// TIA Portal V17 export
// export: Created 2024-09-02T12:50:19.4817416Z, ExportSetting WithDefaults, DisplayName Totally Integrated Automation Portal, DisplayVersion V17, DisplayName TIA Portal Openness, DisplayVersion V17, DisplayName TIA Portal Version Control Interface, DisplayVersion V17, DisplayName STEP 7 Professional, DisplayVersion V17, DisplayName STEP 7 Safety, DisplayVersion V17, DisplayName WinCC Professional, DisplayVersion V17
FUNCTION "AnwFC_Omron_OP70_2" : Void   // FC190, LAD
{ S7_Optimized_Access := 'TRUE' }
VERSION : 0.1
// stored: AutoNumber false, IsIECCheckEnabled false, SetENOAutomatically false, UDAEnableTagReadback false
   VAR_TEMP
      tVKE0 : Bool;
      tVKE1 : Bool;
      tAuto : Bool;
      tHand : Bool;
      Motion_Release : Bool;
      t_dummy : Bool;
      tHmiBld : Bool;
      tHmiEnbl : Bool;
      tCnt : Int;
      tBAmode : Int;
      tHmiScreen : Bool;
      tHmiRelease : Bool;
      i : Int;
   END_VAR
   VAR_TEMP   // added for the SCL form of the ladder/FBD networks
      _w1 : Bool;
   END_VAR
BEGIN

REGION Network 1: ############# Moving Data To DB ###############
END_REGION

REGION Network 2: Copy Output
END_REGION

REGION Network 3: Copy Input
END_REGION

REGION Network 4: ############# Start Up Conditions ###############
END_REGION

REGION Network 5: VKE0/1
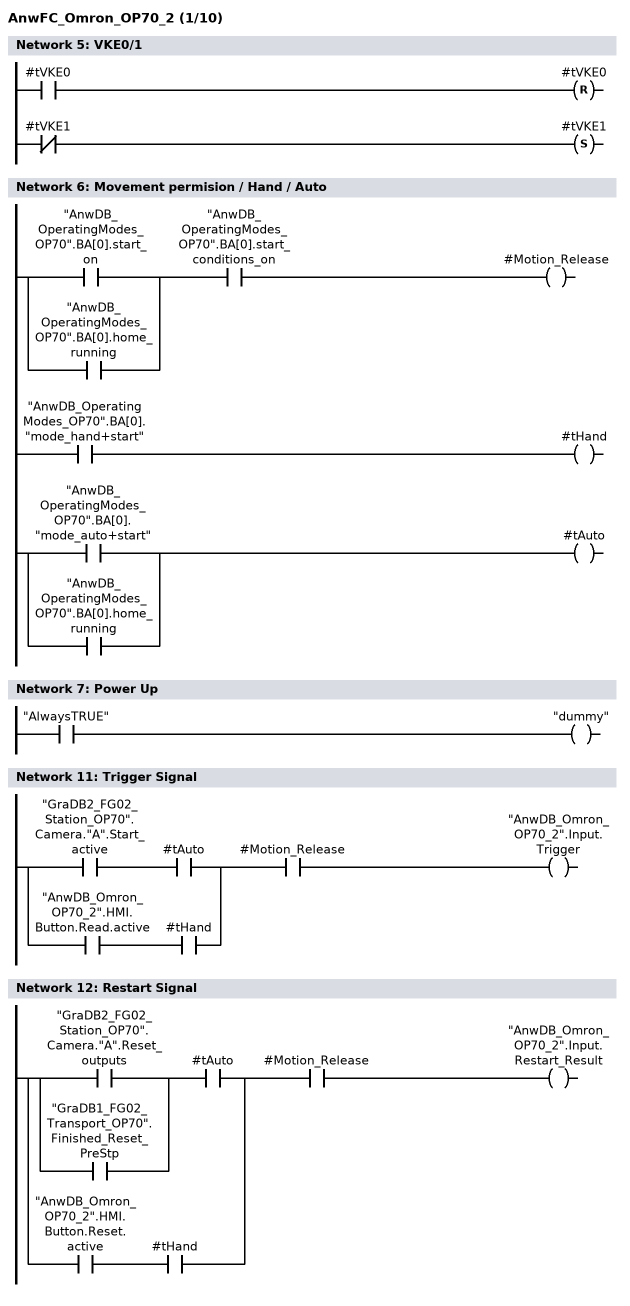
   RUNG wire#powerrail
      Contact( #tVKE0 )
      R_Coil( #tVKE0 )
   END_RUNG
   RUNG wire#powerrail
      I_Contact( #tVKE1 )
      S_Coil( #tVKE1 )
   END_RUNG
   // the same network as SCL:
   IF #tVKE0 THEN #tVKE0 := FALSE; END_IF;
   IF NOT #tVKE1 THEN #tVKE1 := TRUE; END_IF;
END_REGION

REGION Network 6: Movement permision / Hand / Auto
   RUNG wire#powerrail
      Contact( "AnwDB_OperatingModes_OP70".BA[0].start_on )
      wire#w1
      Contact( "AnwDB_OperatingModes_OP70".BA[0].start_conditions_on )
      Coil( #Motion_Release )
   END_RUNG
   RUNG wire#powerrail
      Contact( "AnwDB_OperatingModes_OP70".BA[0].home_running )
   END_RUNG wire#w1
   RUNG wire#powerrail
      Contact( "AnwDB_OperatingModes_OP70".BA[0]."mode_hand+start" )
      Coil( #tHand )
   END_RUNG
   RUNG wire#powerrail
      Contact( "AnwDB_OperatingModes_OP70".BA[0]."mode_auto+start" )
      wire#w2
      Coil( #tAuto )
   END_RUNG
   RUNG wire#powerrail
      Contact( "AnwDB_OperatingModes_OP70".BA[0].home_running )
   END_RUNG wire#w2
   // the same network as SCL:
   #Motion_Release := ("AnwDB_OperatingModes_OP70".BA[0].start_on OR "AnwDB_OperatingModes_OP70".BA[0].home_running) AND "AnwDB_OperatingModes_OP70".BA[0].start_conditions_on;
   #tHand := "AnwDB_OperatingModes_OP70".BA[0]."mode_hand+start";
   #tAuto := "AnwDB_OperatingModes_OP70".BA[0]."mode_auto+start" OR "AnwDB_OperatingModes_OP70".BA[0].home_running;
END_REGION

REGION Network 7: Power Up
   RUNG wire#powerrail
      Contact( "AlwaysTRUE" )
      Coil( "dummy" )
   END_RUNG
   // the same network as SCL:
   "dummy" := "AlwaysTRUE";
END_REGION

REGION Network 8: ############# Data Operation ###############
END_REGION

REGION Network 9: Copy ID number
END_REGION

REGION Network 10: ############# Program Selection And Start ###############
END_REGION

REGION Network 11: Trigger Signal
   RUNG wire#powerrail
      Contact( "GraDB2_FG02_Station_OP70".Camera."A".Start_active )
      Contact( #tAuto )
      wire#w1
      Contact( #Motion_Release )
      Coil( "AnwDB_Omron_OP70_2".Input.Trigger )
   END_RUNG
   RUNG wire#powerrail
      Contact( "AnwDB_Omron_OP70_2".HMI.Button.Read.active )
      Contact( #tHand )
   END_RUNG wire#w1
   // the same network as SCL:
   "AnwDB_Omron_OP70_2".Input.Trigger := (("GraDB2_FG02_Station_OP70".Camera."A".Start_active AND #tAuto) OR ("AnwDB_Omron_OP70_2".HMI.Button.Read.active AND #tHand)) AND #Motion_Release;
END_REGION

REGION Network 12: Restart Signal
   RUNG wire#powerrail
      Contact( "GraDB2_FG02_Station_OP70".Camera."A".Reset_outputs )
      wire#w1
      Contact( #tAuto )
      wire#w2
      Contact( #Motion_Release )
      Coil( "AnwDB_Omron_OP70_2".Input.Restart_Result )
   END_RUNG
   RUNG wire#powerrail
      Contact( "GraDB1_FG02_Transport_OP70".Finished_Reset_PreStp )
   END_RUNG wire#w1
   RUNG wire#powerrail
      Contact( "AnwDB_Omron_OP70_2".HMI.Button.Reset.active )
      Contact( #tHand )
   END_RUNG wire#w2
   // the same network as SCL:
   "AnwDB_Omron_OP70_2".Input.Restart_Result := ((("GraDB2_FG02_Station_OP70".Camera."A".Reset_outputs OR "GraDB1_FG02_Transport_OP70".Finished_Reset_PreStp) AND #tAuto) OR ("AnwDB_Omron_OP70_2".HMI.Button.Reset.active AND #tHand)) AND #Motion_Release;
END_REGION

REGION Network 13: Ack Signal
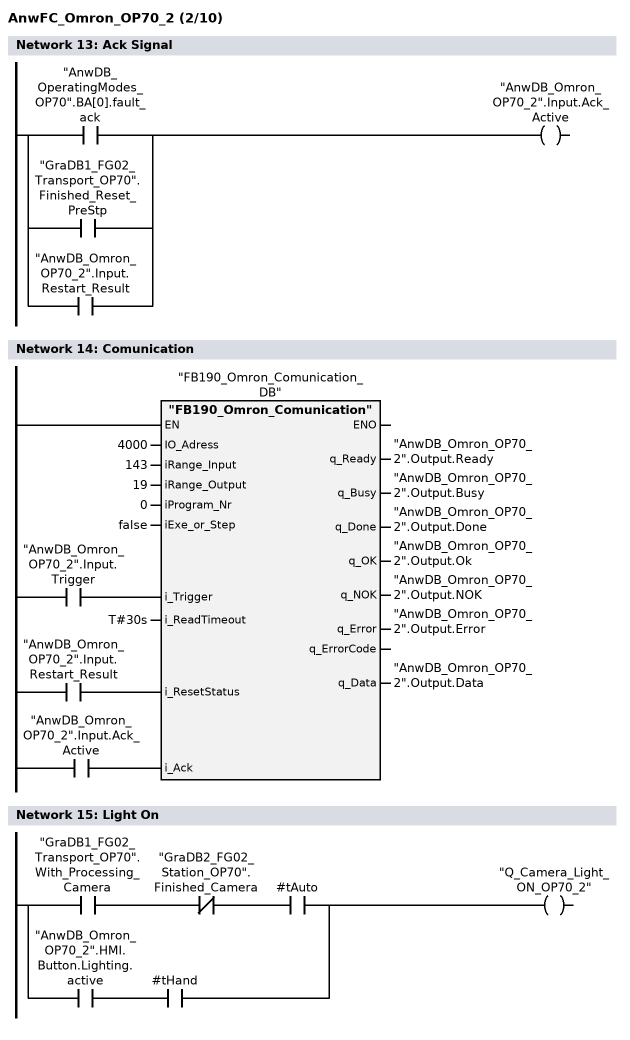
   RUNG wire#powerrail
      Contact( "AnwDB_OperatingModes_OP70".BA[0].fault_ack )
      wire#w1
      Coil( "AnwDB_Omron_OP70_2".Input.Ack_Active )
   END_RUNG
   RUNG wire#powerrail
      Contact( "GraDB1_FG02_Transport_OP70".Finished_Reset_PreStp )
   END_RUNG wire#w1
   RUNG wire#powerrail
      Contact( "AnwDB_Omron_OP70_2".Input.Restart_Result )
   END_RUNG wire#w1
   // the same network as SCL:
   "AnwDB_Omron_OP70_2".Input.Ack_Active := "AnwDB_OperatingModes_OP70".BA[0].fault_ack OR "GraDB1_FG02_Transport_OP70".Finished_Reset_PreStp OR "AnwDB_Omron_OP70_2".Input.Restart_Result;
END_REGION

REGION Network 14: Comunication
   RUNG wire#powerrail
      "FB190_Omron_Comunication_DB"(i_Trigger := wire#w1, i_ResetStatus := wire#w2, i_Ack := wire#w3, IO_Adress := 4000, iRange_Input := 143, iRange_Output := 19, iProgram_Nr := 0, iExe_or_Step := false, i_ReadTimeout := T#30s, q_Ready => "AnwDB_Omron_OP70_2".Output.Ready, q_Busy => "AnwDB_Omron_OP70_2".Output.Busy, q_Done => "AnwDB_Omron_OP70_2".Output.Done, q_OK => "AnwDB_Omron_OP70_2".Output.Ok, q_NOK => "AnwDB_Omron_OP70_2".Output.NOK, q_Error => "AnwDB_Omron_OP70_2".Output.Error, q_ErrorCode =>, q_Data => "AnwDB_Omron_OP70_2".Output.Data)
   END_RUNG
   RUNG wire#powerrail
      Contact( "AnwDB_Omron_OP70_2".Input.Trigger )
   END_RUNG wire#w1
   RUNG wire#powerrail
      Contact( "AnwDB_Omron_OP70_2".Input.Restart_Result )
   END_RUNG wire#w2
   RUNG wire#powerrail
      Contact( "AnwDB_Omron_OP70_2".Input.Ack_Active )
   END_RUNG wire#w3
   // the same network as SCL:
   "FB190_Omron_Comunication_DB"(IO_Adress := 4000,   // "FB190_Omron_Comunication"
                           iRange_Input := 143,
                           iRange_Output := 19,
                           iProgram_Nr := 0,
                           iExe_or_Step := false,
                           i_Trigger := "AnwDB_Omron_OP70_2".Input.Trigger,
                           i_ReadTimeout := T#30s,
                           i_ResetStatus := "AnwDB_Omron_OP70_2".Input.Restart_Result,
                           i_Ack := "AnwDB_Omron_OP70_2".Input.Ack_Active,
                           q_Ready => "AnwDB_Omron_OP70_2".Output.Ready,
                           q_Busy => "AnwDB_Omron_OP70_2".Output.Busy,
                           q_Done => "AnwDB_Omron_OP70_2".Output.Done,
                           q_OK => "AnwDB_Omron_OP70_2".Output.Ok,
                           q_NOK => "AnwDB_Omron_OP70_2".Output.NOK,
                           q_Error => "AnwDB_Omron_OP70_2".Output.Error,
                           q_Data => "AnwDB_Omron_OP70_2".Output.Data);
END_REGION

REGION Network 15: Light On
   RUNG wire#powerrail
      Contact( "GraDB1_FG02_Transport_OP70".With_Processing_Camera )
      I_Contact( "GraDB2_FG02_Station_OP70".Finished_Camera )
      Contact( #tAuto )
      wire#w1
      Coil( "Q_Camera_Light_ON_OP70_2" )
   END_RUNG
   RUNG wire#powerrail
      Contact( "AnwDB_Omron_OP70_2".HMI.Button.Lighting.active )
      Contact( #tHand )
   END_RUNG wire#w1
   // the same network as SCL:
   "Q_Camera_Light_ON_OP70_2" := ("GraDB1_FG02_Transport_OP70".With_Processing_Camera AND NOT "GraDB2_FG02_Station_OP70".Finished_Camera AND #tAuto) OR ("AnwDB_Omron_OP70_2".HMI.Button.Lighting.active AND #tHand);
END_REGION

REGION Network 16: ############# Program Status ###############
END_REGION

REGION Network 17: BEA[1].Ebit[1] - Damper 1 OP 50
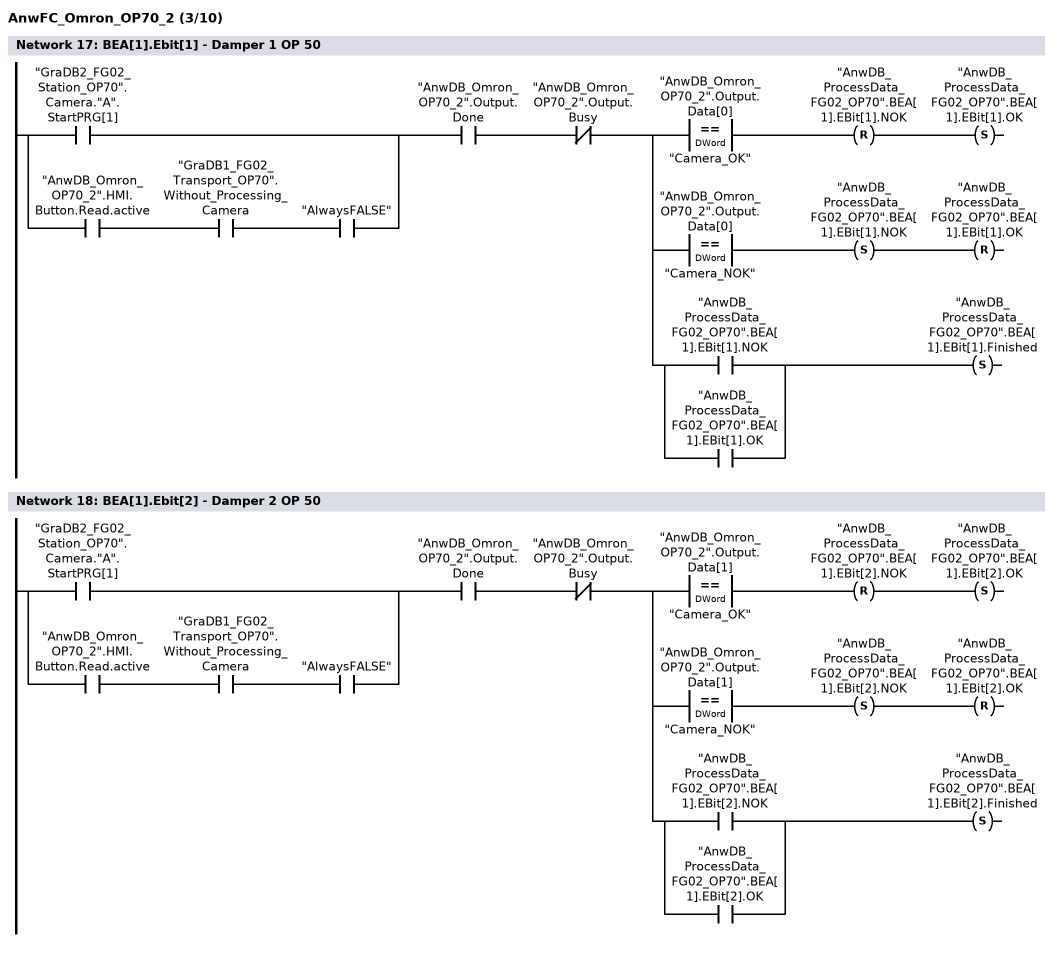
   RUNG wire#powerrail
      Contact( "GraDB2_FG02_Station_OP70".Camera."A".StartPRG[1] )
      wire#w1
      Contact( "AnwDB_Omron_OP70_2".Output.Done )
      I_Contact( "AnwDB_Omron_OP70_2".Output.Busy )
      wire#w2
      { S7_Templates := "SrcType := DWord" } EQ_Contact(in1 := "AnwDB_Omron_OP70_2".Output.Data[0], in2 := "Camera_OK")
      R_Coil( "AnwDB_ProcessData_FG02_OP70".BEA[1].EBit[1].NOK )
      S_Coil( "AnwDB_ProcessData_FG02_OP70".BEA[1].EBit[1].OK )
   END_RUNG
   RUNG wire#powerrail
      Contact( "AnwDB_Omron_OP70_2".HMI.Button.Read.active )
      Contact( "GraDB1_FG02_Transport_OP70".Without_Processing_Camera )
      Contact( "AlwaysFALSE" )
   END_RUNG wire#w1
   RUNG wire#w2
      { S7_Templates := "SrcType := DWord" } EQ_Contact(in1 := "AnwDB_Omron_OP70_2".Output.Data[0], in2 := "Camera_NOK")
      S_Coil( "AnwDB_ProcessData_FG02_OP70".BEA[1].EBit[1].NOK )
      R_Coil( "AnwDB_ProcessData_FG02_OP70".BEA[1].EBit[1].OK )
   END_RUNG
   RUNG wire#w2
      Contact( "AnwDB_ProcessData_FG02_OP70".BEA[1].EBit[1].NOK )
      wire#w3
      S_Coil( "AnwDB_ProcessData_FG02_OP70".BEA[1].EBit[1].Finished )
   END_RUNG
   RUNG wire#w2
      Contact( "AnwDB_ProcessData_FG02_OP70".BEA[1].EBit[1].OK )
   END_RUNG wire#w3
   // the same network as SCL:
   #_w1 := ("GraDB2_FG02_Station_OP70".Camera."A".StartPRG[1] OR ("AnwDB_Omron_OP70_2".HMI.Button.Read.active AND "GraDB1_FG02_Transport_OP70".Without_Processing_Camera AND "AlwaysFALSE")) AND "AnwDB_Omron_OP70_2".Output.Done AND NOT "AnwDB_Omron_OP70_2".Output.Busy;
   IF #_w1 AND ("AnwDB_Omron_OP70_2".Output.Data[0] = "Camera_OK") THEN
       "AnwDB_ProcessData_FG02_OP70".BEA[1].EBit[1].NOK := FALSE;
       "AnwDB_ProcessData_FG02_OP70".BEA[1].EBit[1].OK := TRUE;
   END_IF;
   IF #_w1 AND ("AnwDB_Omron_OP70_2".Output.Data[0] = "Camera_NOK") THEN
       "AnwDB_ProcessData_FG02_OP70".BEA[1].EBit[1].NOK := TRUE;
       "AnwDB_ProcessData_FG02_OP70".BEA[1].EBit[1].OK := FALSE;
   END_IF;
   IF #_w1 AND ("AnwDB_ProcessData_FG02_OP70".BEA[1].EBit[1].NOK OR "AnwDB_ProcessData_FG02_OP70".BEA[1].EBit[1].OK) THEN
       "AnwDB_ProcessData_FG02_OP70".BEA[1].EBit[1].Finished := TRUE;
   END_IF;
END_REGION

REGION Network 18: BEA[1].Ebit[2] - Damper 2 OP 50
   RUNG wire#powerrail
      Contact( "GraDB2_FG02_Station_OP70".Camera."A".StartPRG[1] )
      wire#w1
      Contact( "AnwDB_Omron_OP70_2".Output.Done )
      I_Contact( "AnwDB_Omron_OP70_2".Output.Busy )
      wire#w2
      { S7_Templates := "SrcType := DWord" } EQ_Contact(in1 := "AnwDB_Omron_OP70_2".Output.Data[1], in2 := "Camera_OK")
      R_Coil( "AnwDB_ProcessData_FG02_OP70".BEA[1].EBit[2].NOK )
      S_Coil( "AnwDB_ProcessData_FG02_OP70".BEA[1].EBit[2].OK )
   END_RUNG
   RUNG wire#powerrail
      Contact( "AnwDB_Omron_OP70_2".HMI.Button.Read.active )
      Contact( "GraDB1_FG02_Transport_OP70".Without_Processing_Camera )
      Contact( "AlwaysFALSE" )
   END_RUNG wire#w1
   RUNG wire#w2
      { S7_Templates := "SrcType := DWord" } EQ_Contact(in1 := "AnwDB_Omron_OP70_2".Output.Data[1], in2 := "Camera_NOK")
      S_Coil( "AnwDB_ProcessData_FG02_OP70".BEA[1].EBit[2].NOK )
      R_Coil( "AnwDB_ProcessData_FG02_OP70".BEA[1].EBit[2].OK )
   END_RUNG
   RUNG wire#w2
      Contact( "AnwDB_ProcessData_FG02_OP70".BEA[1].EBit[2].NOK )
      wire#w3
      S_Coil( "AnwDB_ProcessData_FG02_OP70".BEA[1].EBit[2].Finished )
   END_RUNG
   RUNG wire#w2
      Contact( "AnwDB_ProcessData_FG02_OP70".BEA[1].EBit[2].OK )
   END_RUNG wire#w3
   // the same network as SCL:
   #_w1 := ("GraDB2_FG02_Station_OP70".Camera."A".StartPRG[1] OR ("AnwDB_Omron_OP70_2".HMI.Button.Read.active AND "GraDB1_FG02_Transport_OP70".Without_Processing_Camera AND "AlwaysFALSE")) AND "AnwDB_Omron_OP70_2".Output.Done AND NOT "AnwDB_Omron_OP70_2".Output.Busy;
   IF #_w1 AND ("AnwDB_Omron_OP70_2".Output.Data[1] = "Camera_OK") THEN
       "AnwDB_ProcessData_FG02_OP70".BEA[1].EBit[2].NOK := FALSE;
       "AnwDB_ProcessData_FG02_OP70".BEA[1].EBit[2].OK := TRUE;
   END_IF;
   IF #_w1 AND ("AnwDB_Omron_OP70_2".Output.Data[1] = "Camera_NOK") THEN
       "AnwDB_ProcessData_FG02_OP70".BEA[1].EBit[2].NOK := TRUE;
       "AnwDB_ProcessData_FG02_OP70".BEA[1].EBit[2].OK := FALSE;
   END_IF;
   IF #_w1 AND ("AnwDB_ProcessData_FG02_OP70".BEA[1].EBit[2].NOK OR "AnwDB_ProcessData_FG02_OP70".BEA[1].EBit[2].OK) THEN
       "AnwDB_ProcessData_FG02_OP70".BEA[1].EBit[2].Finished := TRUE;
   END_IF;
END_REGION

REGION Network 19: BEA[1].Ebit[3] - Damper 3 OP 50
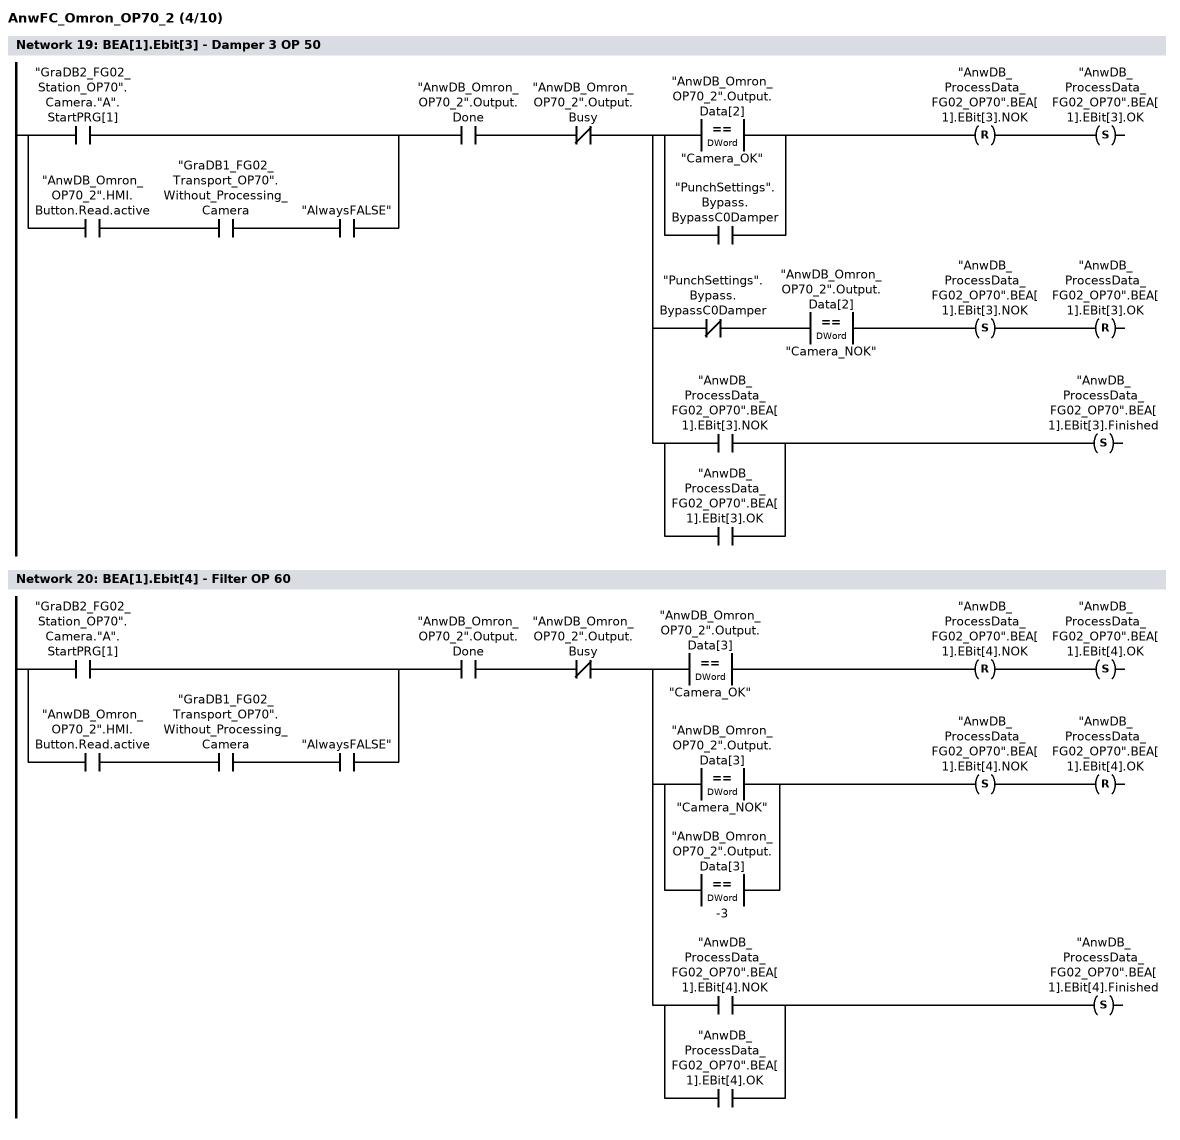
   RUNG wire#powerrail
      Contact( "GraDB2_FG02_Station_OP70".Camera."A".StartPRG[1] )
      wire#w1
      Contact( "AnwDB_Omron_OP70_2".Output.Done )
      I_Contact( "AnwDB_Omron_OP70_2".Output.Busy )
      wire#w2
      { S7_Templates := "SrcType := DWord" } EQ_Contact(in1 := "AnwDB_Omron_OP70_2".Output.Data[2], in2 := "Camera_OK")
      wire#w3
      R_Coil( "AnwDB_ProcessData_FG02_OP70".BEA[1].EBit[3].NOK )
      S_Coil( "AnwDB_ProcessData_FG02_OP70".BEA[1].EBit[3].OK )
   END_RUNG
   RUNG wire#powerrail
      Contact( "AnwDB_Omron_OP70_2".HMI.Button.Read.active )
      Contact( "GraDB1_FG02_Transport_OP70".Without_Processing_Camera )
      Contact( "AlwaysFALSE" )
   END_RUNG wire#w1
   RUNG wire#w2
      Contact( "PunchSettings".Bypass.BypassC0Damper )
   END_RUNG wire#w3
   RUNG wire#w2
      I_Contact( "PunchSettings".Bypass.BypassC0Damper )
      { S7_Templates := "SrcType := DWord" } EQ_Contact(in1 := "AnwDB_Omron_OP70_2".Output.Data[2], in2 := "Camera_NOK")
      S_Coil( "AnwDB_ProcessData_FG02_OP70".BEA[1].EBit[3].NOK )
      R_Coil( "AnwDB_ProcessData_FG02_OP70".BEA[1].EBit[3].OK )
   END_RUNG
   RUNG wire#w2
      Contact( "AnwDB_ProcessData_FG02_OP70".BEA[1].EBit[3].NOK )
      wire#w4
      S_Coil( "AnwDB_ProcessData_FG02_OP70".BEA[1].EBit[3].Finished )
   END_RUNG
   RUNG wire#w2
      Contact( "AnwDB_ProcessData_FG02_OP70".BEA[1].EBit[3].OK )
   END_RUNG wire#w4
   // the same network as SCL:
   #_w1 := ("GraDB2_FG02_Station_OP70".Camera."A".StartPRG[1] OR ("AnwDB_Omron_OP70_2".HMI.Button.Read.active AND "GraDB1_FG02_Transport_OP70".Without_Processing_Camera AND "AlwaysFALSE")) AND "AnwDB_Omron_OP70_2".Output.Done AND NOT "AnwDB_Omron_OP70_2".Output.Busy;
   IF #_w1 AND (("AnwDB_Omron_OP70_2".Output.Data[2] = "Camera_OK") OR "PunchSettings".Bypass.BypassC0Damper) THEN
       "AnwDB_ProcessData_FG02_OP70".BEA[1].EBit[3].NOK := FALSE;
       "AnwDB_ProcessData_FG02_OP70".BEA[1].EBit[3].OK := TRUE;
   END_IF;
   IF #_w1 AND NOT "PunchSettings".Bypass.BypassC0Damper AND ("AnwDB_Omron_OP70_2".Output.Data[2] = "Camera_NOK") THEN
       "AnwDB_ProcessData_FG02_OP70".BEA[1].EBit[3].NOK := TRUE;
       "AnwDB_ProcessData_FG02_OP70".BEA[1].EBit[3].OK := FALSE;
   END_IF;
   IF #_w1 AND ("AnwDB_ProcessData_FG02_OP70".BEA[1].EBit[3].NOK OR "AnwDB_ProcessData_FG02_OP70".BEA[1].EBit[3].OK) THEN
       "AnwDB_ProcessData_FG02_OP70".BEA[1].EBit[3].Finished := TRUE;
   END_IF;
END_REGION

REGION Network 20: BEA[1].Ebit[4] - Filter OP 60
   RUNG wire#powerrail
      Contact( "GraDB2_FG02_Station_OP70".Camera."A".StartPRG[1] )
      wire#w1
      Contact( "AnwDB_Omron_OP70_2".Output.Done )
      I_Contact( "AnwDB_Omron_OP70_2".Output.Busy )
      wire#w2
      { S7_Templates := "SrcType := DWord" } EQ_Contact(in1 := "AnwDB_Omron_OP70_2".Output.Data[3], in2 := "Camera_OK")
      R_Coil( "AnwDB_ProcessData_FG02_OP70".BEA[1].EBit[4].NOK )
      S_Coil( "AnwDB_ProcessData_FG02_OP70".BEA[1].EBit[4].OK )
   END_RUNG
   RUNG wire#powerrail
      Contact( "AnwDB_Omron_OP70_2".HMI.Button.Read.active )
      Contact( "GraDB1_FG02_Transport_OP70".Without_Processing_Camera )
      Contact( "AlwaysFALSE" )
   END_RUNG wire#w1
   RUNG wire#w2
      { S7_Templates := "SrcType := DWord" } EQ_Contact(in1 := "AnwDB_Omron_OP70_2".Output.Data[3], in2 := "Camera_NOK")
      wire#w3
      S_Coil( "AnwDB_ProcessData_FG02_OP70".BEA[1].EBit[4].NOK )
      R_Coil( "AnwDB_ProcessData_FG02_OP70".BEA[1].EBit[4].OK )
   END_RUNG
   RUNG wire#w2
      { S7_Templates := "SrcType := DWord" } EQ_Contact(in1 := "AnwDB_Omron_OP70_2".Output.Data[3], in2 := -3)
   END_RUNG wire#w3
   RUNG wire#w2
      Contact( "AnwDB_ProcessData_FG02_OP70".BEA[1].EBit[4].NOK )
      wire#w4
      S_Coil( "AnwDB_ProcessData_FG02_OP70".BEA[1].EBit[4].Finished )
   END_RUNG
   RUNG wire#w2
      Contact( "AnwDB_ProcessData_FG02_OP70".BEA[1].EBit[4].OK )
   END_RUNG wire#w4
   // the same network as SCL:
   #_w1 := ("GraDB2_FG02_Station_OP70".Camera."A".StartPRG[1] OR ("AnwDB_Omron_OP70_2".HMI.Button.Read.active AND "GraDB1_FG02_Transport_OP70".Without_Processing_Camera AND "AlwaysFALSE")) AND "AnwDB_Omron_OP70_2".Output.Done AND NOT "AnwDB_Omron_OP70_2".Output.Busy;
   IF #_w1 AND ("AnwDB_Omron_OP70_2".Output.Data[3] = "Camera_OK") THEN
       "AnwDB_ProcessData_FG02_OP70".BEA[1].EBit[4].NOK := FALSE;
       "AnwDB_ProcessData_FG02_OP70".BEA[1].EBit[4].OK := TRUE;
   END_IF;
   IF #_w1 AND (("AnwDB_Omron_OP70_2".Output.Data[3] = "Camera_NOK") OR ("AnwDB_Omron_OP70_2".Output.Data[3] = (-3))) THEN
       "AnwDB_ProcessData_FG02_OP70".BEA[1].EBit[4].NOK := TRUE;
       "AnwDB_ProcessData_FG02_OP70".BEA[1].EBit[4].OK := FALSE;
   END_IF;
   IF #_w1 AND ("AnwDB_ProcessData_FG02_OP70".BEA[1].EBit[4].NOK OR "AnwDB_ProcessData_FG02_OP70".BEA[1].EBit[4].OK) THEN
       "AnwDB_ProcessData_FG02_OP70".BEA[1].EBit[4].Finished := TRUE;
   END_IF;
END_REGION

REGION Network 21: BEA[1].Ebit[5] - Ball OP70_1
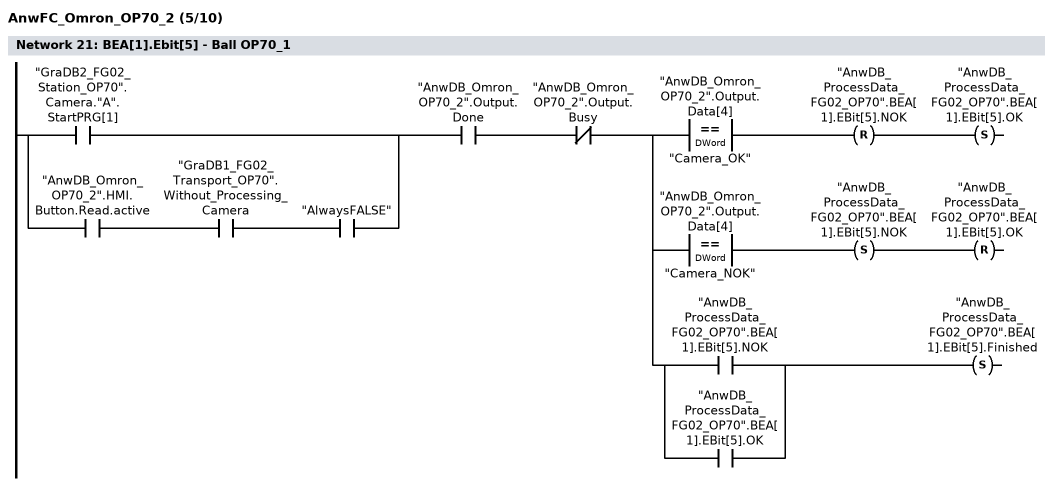
   RUNG wire#powerrail
      Contact( "GraDB2_FG02_Station_OP70".Camera."A".StartPRG[1] )
      wire#w1
      Contact( "AnwDB_Omron_OP70_2".Output.Done )
      I_Contact( "AnwDB_Omron_OP70_2".Output.Busy )
      wire#w2
      { S7_Templates := "SrcType := DWord" } EQ_Contact(in1 := "AnwDB_Omron_OP70_2".Output.Data[4], in2 := "Camera_OK")
      R_Coil( "AnwDB_ProcessData_FG02_OP70".BEA[1].EBit[5].NOK )
      S_Coil( "AnwDB_ProcessData_FG02_OP70".BEA[1].EBit[5].OK )
   END_RUNG
   RUNG wire#powerrail
      Contact( "AnwDB_Omron_OP70_2".HMI.Button.Read.active )
      Contact( "GraDB1_FG02_Transport_OP70".Without_Processing_Camera )
      Contact( "AlwaysFALSE" )
   END_RUNG wire#w1
   RUNG wire#w2
      { S7_Templates := "SrcType := DWord" } EQ_Contact(in1 := "AnwDB_Omron_OP70_2".Output.Data[4], in2 := "Camera_NOK")
      S_Coil( "AnwDB_ProcessData_FG02_OP70".BEA[1].EBit[5].NOK )
      R_Coil( "AnwDB_ProcessData_FG02_OP70".BEA[1].EBit[5].OK )
   END_RUNG
   RUNG wire#w2
      Contact( "AnwDB_ProcessData_FG02_OP70".BEA[1].EBit[5].NOK )
      wire#w3
      S_Coil( "AnwDB_ProcessData_FG02_OP70".BEA[1].EBit[5].Finished )
   END_RUNG
   RUNG wire#w2
      Contact( "AnwDB_ProcessData_FG02_OP70".BEA[1].EBit[5].OK )
   END_RUNG wire#w3
   // the same network as SCL:
   #_w1 := ("GraDB2_FG02_Station_OP70".Camera."A".StartPRG[1] OR ("AnwDB_Omron_OP70_2".HMI.Button.Read.active AND "GraDB1_FG02_Transport_OP70".Without_Processing_Camera AND "AlwaysFALSE")) AND "AnwDB_Omron_OP70_2".Output.Done AND NOT "AnwDB_Omron_OP70_2".Output.Busy;
   IF #_w1 AND ("AnwDB_Omron_OP70_2".Output.Data[4] = "Camera_OK") THEN
       "AnwDB_ProcessData_FG02_OP70".BEA[1].EBit[5].NOK := FALSE;
       "AnwDB_ProcessData_FG02_OP70".BEA[1].EBit[5].OK := TRUE;
   END_IF;
   IF #_w1 AND ("AnwDB_Omron_OP70_2".Output.Data[4] = "Camera_NOK") THEN
       "AnwDB_ProcessData_FG02_OP70".BEA[1].EBit[5].NOK := TRUE;
       "AnwDB_ProcessData_FG02_OP70".BEA[1].EBit[5].OK := FALSE;
   END_IF;
   IF #_w1 AND ("AnwDB_ProcessData_FG02_OP70".BEA[1].EBit[5].NOK OR "AnwDB_ProcessData_FG02_OP70".BEA[1].EBit[5].OK) THEN
       "AnwDB_ProcessData_FG02_OP70".BEA[1].EBit[5].Finished := TRUE;
   END_IF;
END_REGION

REGION Network 22: BEA[1].Ebit[6] - Damper Cap OP70_1
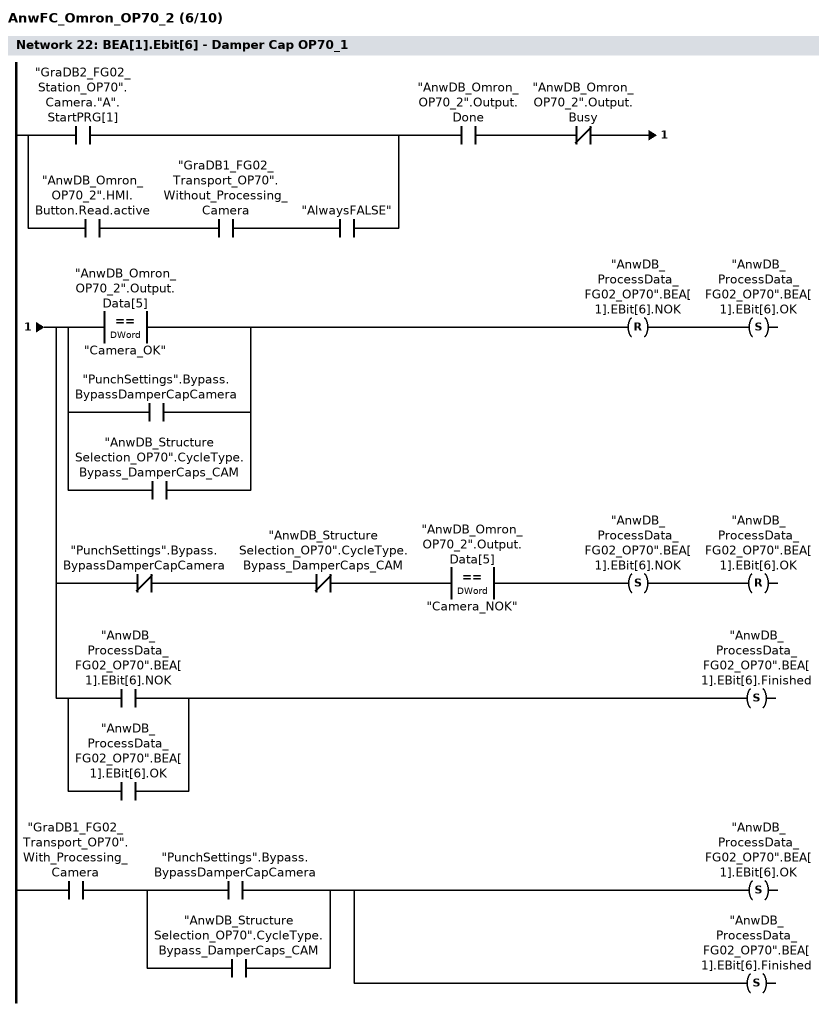
   RUNG wire#powerrail
      Contact( "GraDB2_FG02_Station_OP70".Camera."A".StartPRG[1] )
      wire#w1
      Contact( "AnwDB_Omron_OP70_2".Output.Done )
      I_Contact( "AnwDB_Omron_OP70_2".Output.Busy )
      wire#w2
      { S7_Templates := "SrcType := DWord" } EQ_Contact(in1 := "AnwDB_Omron_OP70_2".Output.Data[5], in2 := "Camera_OK")
      wire#w3
      R_Coil( "AnwDB_ProcessData_FG02_OP70".BEA[1].EBit[6].NOK )
      S_Coil( "AnwDB_ProcessData_FG02_OP70".BEA[1].EBit[6].OK )
   END_RUNG
   RUNG wire#powerrail
      Contact( "AnwDB_Omron_OP70_2".HMI.Button.Read.active )
      Contact( "GraDB1_FG02_Transport_OP70".Without_Processing_Camera )
      Contact( "AlwaysFALSE" )
   END_RUNG wire#w1
   RUNG wire#w2
      Contact( "PunchSettings".Bypass.BypassDamperCapCamera )
   END_RUNG wire#w3
   RUNG wire#w2
      Contact( "AnwDB_StructureSelection_OP70".CycleType.Bypass_DamperCaps_CAM )
   END_RUNG wire#w3
   RUNG wire#w2
      I_Contact( "PunchSettings".Bypass.BypassDamperCapCamera )
      I_Contact( "AnwDB_StructureSelection_OP70".CycleType.Bypass_DamperCaps_CAM )
      { S7_Templates := "SrcType := DWord" } EQ_Contact(in1 := "AnwDB_Omron_OP70_2".Output.Data[5], in2 := "Camera_NOK")
      S_Coil( "AnwDB_ProcessData_FG02_OP70".BEA[1].EBit[6].NOK )
      R_Coil( "AnwDB_ProcessData_FG02_OP70".BEA[1].EBit[6].OK )
   END_RUNG
   RUNG wire#w2
      Contact( "AnwDB_ProcessData_FG02_OP70".BEA[1].EBit[6].NOK )
      wire#w4
      S_Coil( "AnwDB_ProcessData_FG02_OP70".BEA[1].EBit[6].Finished )
   END_RUNG
   RUNG wire#w2
      Contact( "AnwDB_ProcessData_FG02_OP70".BEA[1].EBit[6].OK )
   END_RUNG wire#w4
   RUNG wire#powerrail
      Contact( "GraDB1_FG02_Transport_OP70".With_Processing_Camera )
      wire#w5
      Contact( "PunchSettings".Bypass.BypassDamperCapCamera )
      wire#w6
      S_Coil( "AnwDB_ProcessData_FG02_OP70".BEA[1].EBit[6].OK )
   END_RUNG
   RUNG wire#w5
      Contact( "AnwDB_StructureSelection_OP70".CycleType.Bypass_DamperCaps_CAM )
   END_RUNG wire#w6
   RUNG wire#w6
      S_Coil( "AnwDB_ProcessData_FG02_OP70".BEA[1].EBit[6].Finished )
   END_RUNG
   // the same network as SCL:
   #_w1 := ("GraDB2_FG02_Station_OP70".Camera."A".StartPRG[1] OR ("AnwDB_Omron_OP70_2".HMI.Button.Read.active AND "GraDB1_FG02_Transport_OP70".Without_Processing_Camera AND "AlwaysFALSE")) AND "AnwDB_Omron_OP70_2".Output.Done AND NOT "AnwDB_Omron_OP70_2".Output.Busy;
   IF #_w1 AND (("AnwDB_Omron_OP70_2".Output.Data[5] = "Camera_OK") OR "PunchSettings".Bypass.BypassDamperCapCamera OR "AnwDB_StructureSelection_OP70".CycleType.Bypass_DamperCaps_CAM) THEN
       "AnwDB_ProcessData_FG02_OP70".BEA[1].EBit[6].NOK := FALSE;
       "AnwDB_ProcessData_FG02_OP70".BEA[1].EBit[6].OK := TRUE;
   END_IF;
   IF #_w1 AND NOT "PunchSettings".Bypass.BypassDamperCapCamera AND NOT "AnwDB_StructureSelection_OP70".CycleType.Bypass_DamperCaps_CAM AND ("AnwDB_Omron_OP70_2".Output.Data[5] = "Camera_NOK") THEN
       "AnwDB_ProcessData_FG02_OP70".BEA[1].EBit[6].NOK := TRUE;
       "AnwDB_ProcessData_FG02_OP70".BEA[1].EBit[6].OK := FALSE;
   END_IF;
   IF #_w1 AND ("AnwDB_ProcessData_FG02_OP70".BEA[1].EBit[6].NOK OR "AnwDB_ProcessData_FG02_OP70".BEA[1].EBit[6].OK) THEN
       "AnwDB_ProcessData_FG02_OP70".BEA[1].EBit[6].Finished := TRUE;
   END_IF;
   IF "GraDB1_FG02_Transport_OP70".With_Processing_Camera AND ("PunchSettings".Bypass.BypassDamperCapCamera OR "AnwDB_StructureSelection_OP70".CycleType.Bypass_DamperCaps_CAM) THEN
       "AnwDB_ProcessData_FG02_OP70".BEA[1].EBit[6].OK := TRUE;
       "AnwDB_ProcessData_FG02_OP70".BEA[1].EBit[6].Finished := TRUE;
   END_IF;
END_REGION

REGION Network 23: BEA[1].Ebit[7] - Dowel 1 OP60
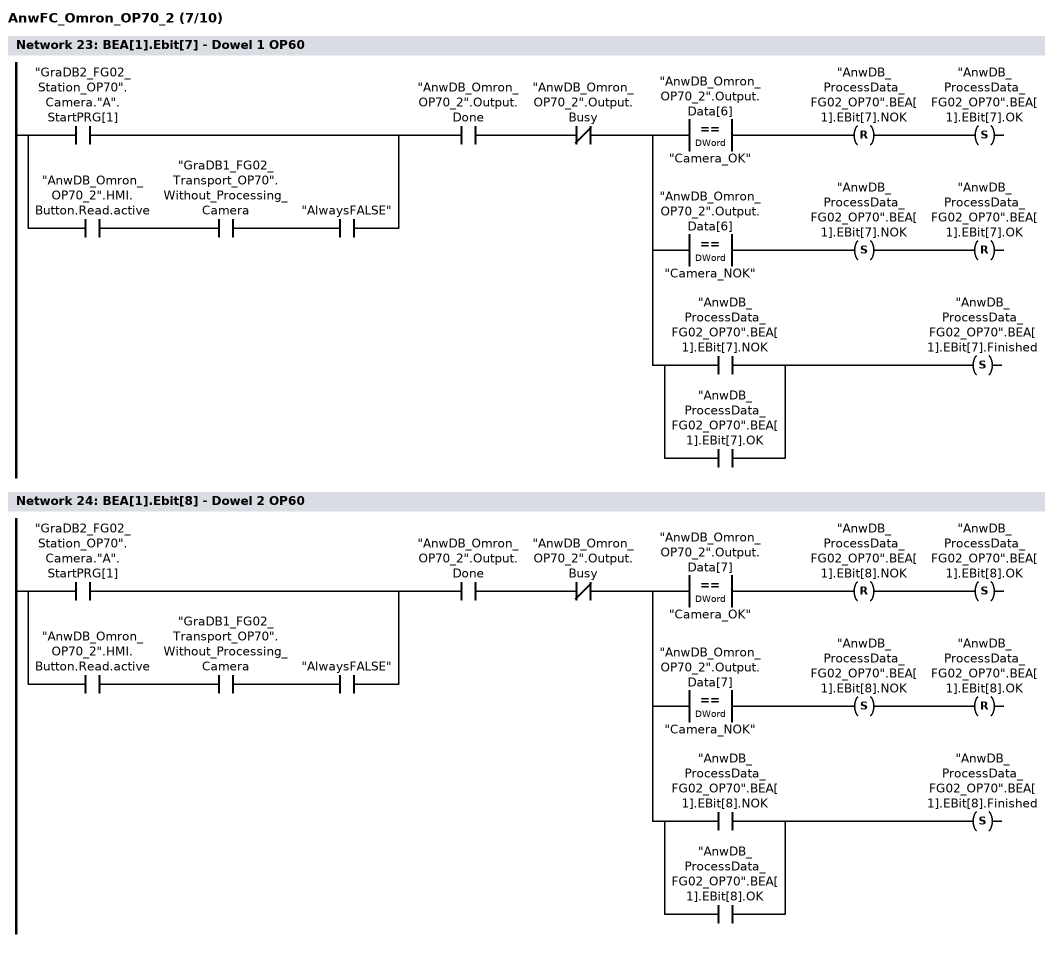
   RUNG wire#powerrail
      Contact( "GraDB2_FG02_Station_OP70".Camera."A".StartPRG[1] )
      wire#w1
      Contact( "AnwDB_Omron_OP70_2".Output.Done )
      I_Contact( "AnwDB_Omron_OP70_2".Output.Busy )
      wire#w2
      { S7_Templates := "SrcType := DWord" } EQ_Contact(in1 := "AnwDB_Omron_OP70_2".Output.Data[6], in2 := "Camera_OK")
      R_Coil( "AnwDB_ProcessData_FG02_OP70".BEA[1].EBit[7].NOK )
      S_Coil( "AnwDB_ProcessData_FG02_OP70".BEA[1].EBit[7].OK )
   END_RUNG
   RUNG wire#powerrail
      Contact( "AnwDB_Omron_OP70_2".HMI.Button.Read.active )
      Contact( "GraDB1_FG02_Transport_OP70".Without_Processing_Camera )
      Contact( "AlwaysFALSE" )
   END_RUNG wire#w1
   RUNG wire#w2
      { S7_Templates := "SrcType := DWord" } EQ_Contact(in1 := "AnwDB_Omron_OP70_2".Output.Data[6], in2 := "Camera_NOK")
      S_Coil( "AnwDB_ProcessData_FG02_OP70".BEA[1].EBit[7].NOK )
      R_Coil( "AnwDB_ProcessData_FG02_OP70".BEA[1].EBit[7].OK )
   END_RUNG
   RUNG wire#w2
      Contact( "AnwDB_ProcessData_FG02_OP70".BEA[1].EBit[7].NOK )
      wire#w3
      S_Coil( "AnwDB_ProcessData_FG02_OP70".BEA[1].EBit[7].Finished )
   END_RUNG
   RUNG wire#w2
      Contact( "AnwDB_ProcessData_FG02_OP70".BEA[1].EBit[7].OK )
   END_RUNG wire#w3
   // the same network as SCL:
   #_w1 := ("GraDB2_FG02_Station_OP70".Camera."A".StartPRG[1] OR ("AnwDB_Omron_OP70_2".HMI.Button.Read.active AND "GraDB1_FG02_Transport_OP70".Without_Processing_Camera AND "AlwaysFALSE")) AND "AnwDB_Omron_OP70_2".Output.Done AND NOT "AnwDB_Omron_OP70_2".Output.Busy;
   IF #_w1 AND ("AnwDB_Omron_OP70_2".Output.Data[6] = "Camera_OK") THEN
       "AnwDB_ProcessData_FG02_OP70".BEA[1].EBit[7].NOK := FALSE;
       "AnwDB_ProcessData_FG02_OP70".BEA[1].EBit[7].OK := TRUE;
   END_IF;
   IF #_w1 AND ("AnwDB_Omron_OP70_2".Output.Data[6] = "Camera_NOK") THEN
       "AnwDB_ProcessData_FG02_OP70".BEA[1].EBit[7].NOK := TRUE;
       "AnwDB_ProcessData_FG02_OP70".BEA[1].EBit[7].OK := FALSE;
   END_IF;
   IF #_w1 AND ("AnwDB_ProcessData_FG02_OP70".BEA[1].EBit[7].NOK OR "AnwDB_ProcessData_FG02_OP70".BEA[1].EBit[7].OK) THEN
       "AnwDB_ProcessData_FG02_OP70".BEA[1].EBit[7].Finished := TRUE;
   END_IF;
END_REGION

REGION Network 24: BEA[1].Ebit[8] - Dowel 2 OP60
   RUNG wire#powerrail
      Contact( "GraDB2_FG02_Station_OP70".Camera."A".StartPRG[1] )
      wire#w1
      Contact( "AnwDB_Omron_OP70_2".Output.Done )
      I_Contact( "AnwDB_Omron_OP70_2".Output.Busy )
      wire#w2
      { S7_Templates := "SrcType := DWord" } EQ_Contact(in1 := "AnwDB_Omron_OP70_2".Output.Data[7], in2 := "Camera_OK")
      R_Coil( "AnwDB_ProcessData_FG02_OP70".BEA[1].EBit[8].NOK )
      S_Coil( "AnwDB_ProcessData_FG02_OP70".BEA[1].EBit[8].OK )
   END_RUNG
   RUNG wire#powerrail
      Contact( "AnwDB_Omron_OP70_2".HMI.Button.Read.active )
      Contact( "GraDB1_FG02_Transport_OP70".Without_Processing_Camera )
      Contact( "AlwaysFALSE" )
   END_RUNG wire#w1
   RUNG wire#w2
      { S7_Templates := "SrcType := DWord" } EQ_Contact(in1 := "AnwDB_Omron_OP70_2".Output.Data[7], in2 := "Camera_NOK")
      S_Coil( "AnwDB_ProcessData_FG02_OP70".BEA[1].EBit[8].NOK )
      R_Coil( "AnwDB_ProcessData_FG02_OP70".BEA[1].EBit[8].OK )
   END_RUNG
   RUNG wire#w2
      Contact( "AnwDB_ProcessData_FG02_OP70".BEA[1].EBit[8].NOK )
      wire#w3
      S_Coil( "AnwDB_ProcessData_FG02_OP70".BEA[1].EBit[8].Finished )
   END_RUNG
   RUNG wire#w2
      Contact( "AnwDB_ProcessData_FG02_OP70".BEA[1].EBit[8].OK )
   END_RUNG wire#w3
   // the same network as SCL:
   #_w1 := ("GraDB2_FG02_Station_OP70".Camera."A".StartPRG[1] OR ("AnwDB_Omron_OP70_2".HMI.Button.Read.active AND "GraDB1_FG02_Transport_OP70".Without_Processing_Camera AND "AlwaysFALSE")) AND "AnwDB_Omron_OP70_2".Output.Done AND NOT "AnwDB_Omron_OP70_2".Output.Busy;
   IF #_w1 AND ("AnwDB_Omron_OP70_2".Output.Data[7] = "Camera_OK") THEN
       "AnwDB_ProcessData_FG02_OP70".BEA[1].EBit[8].NOK := FALSE;
       "AnwDB_ProcessData_FG02_OP70".BEA[1].EBit[8].OK := TRUE;
   END_IF;
   IF #_w1 AND ("AnwDB_Omron_OP70_2".Output.Data[7] = "Camera_NOK") THEN
       "AnwDB_ProcessData_FG02_OP70".BEA[1].EBit[8].NOK := TRUE;
       "AnwDB_ProcessData_FG02_OP70".BEA[1].EBit[8].OK := FALSE;
   END_IF;
   IF #_w1 AND ("AnwDB_ProcessData_FG02_OP70".BEA[1].EBit[8].NOK OR "AnwDB_ProcessData_FG02_OP70".BEA[1].EBit[8].OK) THEN
       "AnwDB_ProcessData_FG02_OP70".BEA[1].EBit[8].Finished := TRUE;
   END_IF;
END_REGION

REGION Network 25: BEA - Started bit
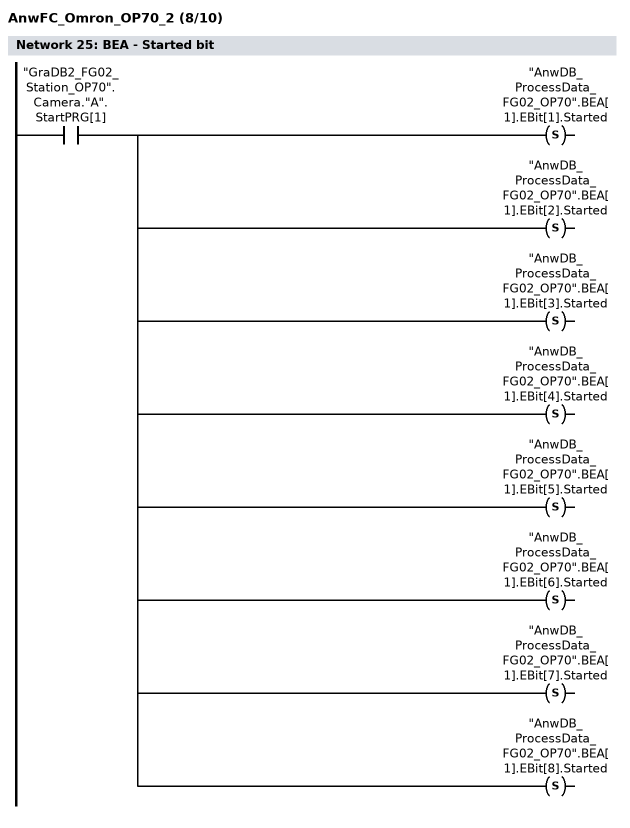
   RUNG wire#powerrail
      Contact( "GraDB2_FG02_Station_OP70".Camera."A".StartPRG[1] )
      wire#w1
      S_Coil( "AnwDB_ProcessData_FG02_OP70".BEA[1].EBit[1].Started )
   END_RUNG
   RUNG wire#w1
      S_Coil( "AnwDB_ProcessData_FG02_OP70".BEA[1].EBit[2].Started )
   END_RUNG
   RUNG wire#w1
      S_Coil( "AnwDB_ProcessData_FG02_OP70".BEA[1].EBit[3].Started )
   END_RUNG
   RUNG wire#w1
      S_Coil( "AnwDB_ProcessData_FG02_OP70".BEA[1].EBit[4].Started )
   END_RUNG
   RUNG wire#w1
      S_Coil( "AnwDB_ProcessData_FG02_OP70".BEA[1].EBit[5].Started )
   END_RUNG
   RUNG wire#w1
      S_Coil( "AnwDB_ProcessData_FG02_OP70".BEA[1].EBit[6].Started )
   END_RUNG
   RUNG wire#w1
      S_Coil( "AnwDB_ProcessData_FG02_OP70".BEA[1].EBit[7].Started )
   END_RUNG
   RUNG wire#w1
      S_Coil( "AnwDB_ProcessData_FG02_OP70".BEA[1].EBit[8].Started )
   END_RUNG
   // the same network as SCL:
   IF "GraDB2_FG02_Station_OP70".Camera."A".StartPRG[1] THEN
       "AnwDB_ProcessData_FG02_OP70".BEA[1].EBit[1].Started := TRUE;
       "AnwDB_ProcessData_FG02_OP70".BEA[1].EBit[2].Started := TRUE;
       "AnwDB_ProcessData_FG02_OP70".BEA[1].EBit[3].Started := TRUE;
       "AnwDB_ProcessData_FG02_OP70".BEA[1].EBit[4].Started := TRUE;
       "AnwDB_ProcessData_FG02_OP70".BEA[1].EBit[5].Started := TRUE;
       "AnwDB_ProcessData_FG02_OP70".BEA[1].EBit[6].Started := TRUE;
       "AnwDB_ProcessData_FG02_OP70".BEA[1].EBit[7].Started := TRUE;
       "AnwDB_ProcessData_FG02_OP70".BEA[1].EBit[8].Started := TRUE;
   END_IF;
END_REGION

REGION Network 26: HMI Result
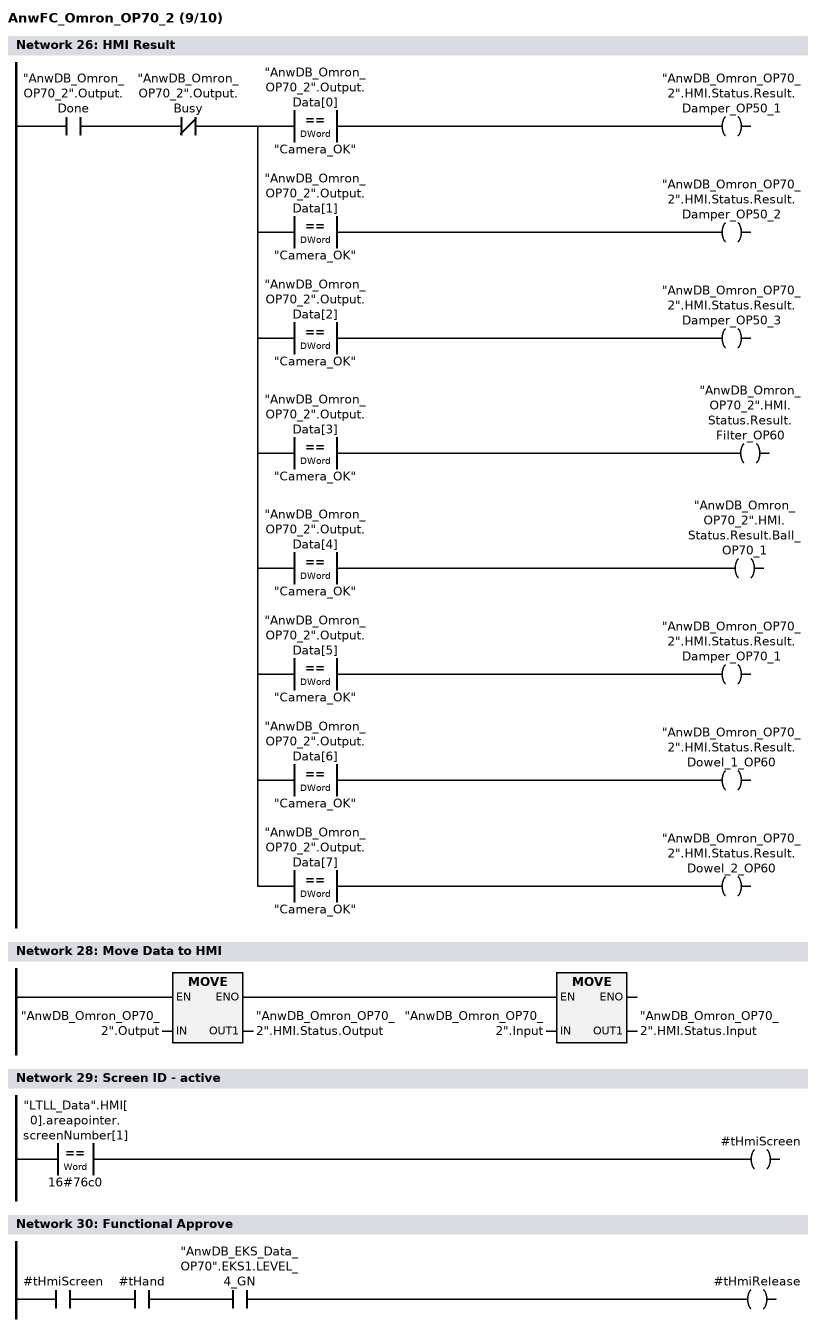
   RUNG wire#powerrail
      Contact( "AnwDB_Omron_OP70_2".Output.Done )
      I_Contact( "AnwDB_Omron_OP70_2".Output.Busy )
      wire#w1
      { S7_Templates := "SrcType := DWord" } EQ_Contact(in1 := "AnwDB_Omron_OP70_2".Output.Data[0], in2 := "Camera_OK")
      Coil( "AnwDB_Omron_OP70_2".HMI.Status.Result.Damper_OP50_1 )
   END_RUNG
   RUNG wire#w1
      { S7_Templates := "SrcType := DWord" } EQ_Contact(in1 := "AnwDB_Omron_OP70_2".Output.Data[1], in2 := "Camera_OK")
      Coil( "AnwDB_Omron_OP70_2".HMI.Status.Result.Damper_OP50_2 )
   END_RUNG
   RUNG wire#w1
      { S7_Templates := "SrcType := DWord" } EQ_Contact(in1 := "AnwDB_Omron_OP70_2".Output.Data[2], in2 := "Camera_OK")
      Coil( "AnwDB_Omron_OP70_2".HMI.Status.Result.Damper_OP50_3 )
   END_RUNG
   RUNG wire#w1
      { S7_Templates := "SrcType := DWord" } EQ_Contact(in1 := "AnwDB_Omron_OP70_2".Output.Data[3], in2 := "Camera_OK")
      Coil( "AnwDB_Omron_OP70_2".HMI.Status.Result.Filter_OP60 )
   END_RUNG
   RUNG wire#w1
      { S7_Templates := "SrcType := DWord" } EQ_Contact(in1 := "AnwDB_Omron_OP70_2".Output.Data[4], in2 := "Camera_OK")
      Coil( "AnwDB_Omron_OP70_2".HMI.Status.Result.Ball_OP70_1 )
   END_RUNG
   RUNG wire#w1
      { S7_Templates := "SrcType := DWord" } EQ_Contact(in1 := "AnwDB_Omron_OP70_2".Output.Data[5], in2 := "Camera_OK")
      Coil( "AnwDB_Omron_OP70_2".HMI.Status.Result.Damper_OP70_1 )
   END_RUNG
   RUNG wire#w1
      { S7_Templates := "SrcType := DWord" } EQ_Contact(in1 := "AnwDB_Omron_OP70_2".Output.Data[6], in2 := "Camera_OK")
      Coil( "AnwDB_Omron_OP70_2".HMI.Status.Result.Dowel_1_OP60 )
   END_RUNG
   RUNG wire#w1
      { S7_Templates := "SrcType := DWord" } EQ_Contact(in1 := "AnwDB_Omron_OP70_2".Output.Data[7], in2 := "Camera_OK")
      Coil( "AnwDB_Omron_OP70_2".HMI.Status.Result.Dowel_2_OP60 )
   END_RUNG
   // the same network as SCL:
   #_w1 := "AnwDB_Omron_OP70_2".Output.Done AND NOT "AnwDB_Omron_OP70_2".Output.Busy;
   "AnwDB_Omron_OP70_2".HMI.Status.Result.Damper_OP50_1 := #_w1 AND ("AnwDB_Omron_OP70_2".Output.Data[0] = "Camera_OK");
   "AnwDB_Omron_OP70_2".HMI.Status.Result.Damper_OP50_2 := #_w1 AND ("AnwDB_Omron_OP70_2".Output.Data[1] = "Camera_OK");
   "AnwDB_Omron_OP70_2".HMI.Status.Result.Damper_OP50_3 := #_w1 AND ("AnwDB_Omron_OP70_2".Output.Data[2] = "Camera_OK");
   "AnwDB_Omron_OP70_2".HMI.Status.Result.Filter_OP60 := #_w1 AND ("AnwDB_Omron_OP70_2".Output.Data[3] = "Camera_OK");
   "AnwDB_Omron_OP70_2".HMI.Status.Result.Ball_OP70_1 := #_w1 AND ("AnwDB_Omron_OP70_2".Output.Data[4] = "Camera_OK");
   "AnwDB_Omron_OP70_2".HMI.Status.Result.Damper_OP70_1 := #_w1 AND ("AnwDB_Omron_OP70_2".Output.Data[5] = "Camera_OK");
   "AnwDB_Omron_OP70_2".HMI.Status.Result.Dowel_1_OP60 := #_w1 AND ("AnwDB_Omron_OP70_2".Output.Data[6] = "Camera_OK");
   "AnwDB_Omron_OP70_2".HMI.Status.Result.Dowel_2_OP60 := #_w1 AND ("AnwDB_Omron_OP70_2".Output.Data[7] = "Camera_OK");
END_REGION

REGION Network 27: ############## HMI #############
END_REGION

REGION Network 28: Move Data to HMI
   RUNG wire#powerrail
      Move(in := "AnwDB_Omron_OP70_2".Output, out1 => "AnwDB_Omron_OP70_2".HMI.Status.Output)
      Move(in := "AnwDB_Omron_OP70_2".Input, out1 => "AnwDB_Omron_OP70_2".HMI.Status.Input)
   END_RUNG
   // the same network as SCL:
   "AnwDB_Omron_OP70_2".HMI.Status.Output := "AnwDB_Omron_OP70_2".Output;
   "AnwDB_Omron_OP70_2".HMI.Status.Input := "AnwDB_Omron_OP70_2".Input;
END_REGION

REGION Network 29: Screen ID - active
   RUNG wire#powerrail
      { S7_Templates := "SrcType := Word" } EQ_Contact(in1 := "LTLL_Data".HMI[0].areapointer.screenNumber[1], in2 := 16#76c0)
      Coil( #tHmiScreen )
   END_RUNG
   // the same network as SCL:
   #tHmiScreen := "LTLL_Data".HMI[0].areapointer.screenNumber[1] = 16#76c0;
END_REGION

REGION Network 30: Functional Approve
   RUNG wire#powerrail
      Contact( #tHmiScreen )
      Contact( #tHand )
      Contact( "AnwDB_EKS_Data_OP70".EKS1.LEVEL_4_GN )
      Coil( #tHmiRelease )
   END_RUNG
   // the same network as SCL:
   #tHmiRelease := #tHmiScreen AND #tHand AND "AnwDB_EKS_Data_OP70".EKS1.LEVEL_4_GN;
END_REGION

REGION Network 31: Functional Approve
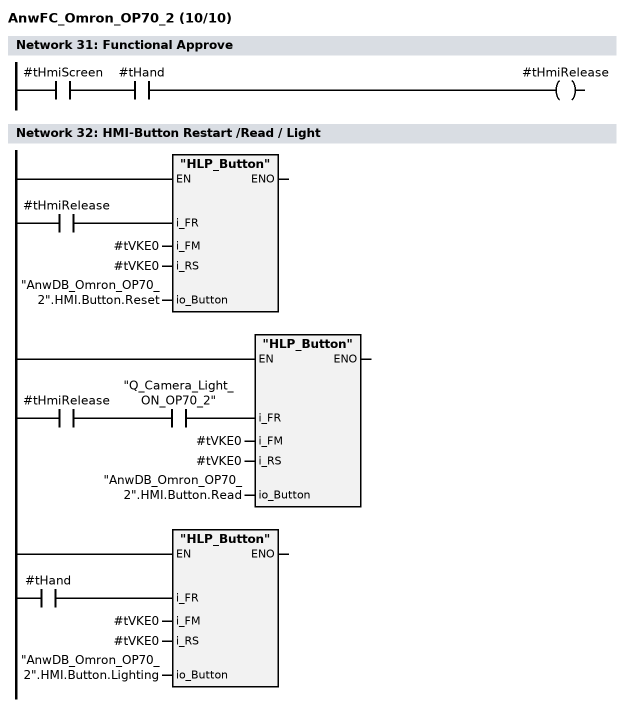
   RUNG wire#powerrail
      Contact( #tHmiScreen )
      Contact( #tHand )
      Coil( #tHmiRelease )
   END_RUNG
   // the same network as SCL:
   #tHmiRelease := #tHmiScreen AND #tHand;
END_REGION

REGION Network 32: HMI-Button Restart /Read / Light
   RUNG wire#powerrail
      "HLP_Button"(i_FR := wire#w1, i_FM := #tVKE0, i_RS := #tVKE0, io_Button := "AnwDB_Omron_OP70_2".HMI.Button.Reset)
   END_RUNG
   RUNG wire#powerrail
      Contact( #tHmiRelease )
   END_RUNG wire#w1
   RUNG wire#powerrail
      "HLP_Button"(i_FR := wire#w2, i_FM := #tVKE0, i_RS := #tVKE0, io_Button := "AnwDB_Omron_OP70_2".HMI.Button.Read)
   END_RUNG
   RUNG wire#powerrail
      Contact( #tHmiRelease )
      Contact( "Q_Camera_Light_ON_OP70_2" )
   END_RUNG wire#w2
   RUNG wire#powerrail
      "HLP_Button"(i_FR := wire#w3, i_FM := #tVKE0, i_RS := #tVKE0, io_Button := "AnwDB_Omron_OP70_2".HMI.Button.Lighting)
   END_RUNG
   RUNG wire#powerrail
      Contact( #tHand )
   END_RUNG wire#w3
   // the same network as SCL:
   "HLP_Button"(i_FR := #tHmiRelease,
                i_FM := #tVKE0,
                i_RS := #tVKE0,
                io_Button := "AnwDB_Omron_OP70_2".HMI.Button.Reset);
   "HLP_Button"(i_FR := #tHmiRelease AND "Q_Camera_Light_ON_OP70_2",
                i_FM := #tVKE0,
                i_RS := #tVKE0,
                io_Button := "AnwDB_Omron_OP70_2".HMI.Button.Read);
   "HLP_Button"(i_FR := #tHand,
                i_FM := #tVKE0,
                i_RS := #tVKE0,
                io_Button := "AnwDB_Omron_OP70_2".HMI.Button.Lighting);
END_REGION
END_FUNCTION
